% RSLogix 500 project P7_KOBIERSKI_M.RSS, saved by version 8.30.00.16 %
PROJECT "UNTITLED"    % processor: Bul.1763 MicroLogix 1100 Series B %

PROGRAM FILES
  LAD 2 "MAIN"  4 rungs
  LAD 3 "IO"  6 rungs
  LAD 4 "CYCLE"  5 rungs
  LAD 5 "CALIBRATE"  15 rungs
  LAD 6 "SAMPLE"  7 rungs
  LAD 7 "0% SAMPLE"  7 rungs
  LAD 8 "30% SAMPLE"  7 rungs
  LAD 9 "CALIB CALC"  6 rungs

DATA FILES
  O0 OUTPUT  4 elements
  I1 INPUT  6 elements
  S2 STATUS  66 elements
  B3 BINARY  3 elements
  T4 TIMER  5 elements
  C5 COUNTER  1 elements
  R6 CONTROL  1 elements
  N7 INTEGER  9 elements
  F8 FLOAT  3 elements
  F9 O2 SAMPLES  10 elements
  N10 SAMP STTNG  6 elements
  F11 AVGS  9 elements
  F12 0% SAMPLES  5 elements
  F13 30% SAMPLE  5 elements
  F14 CALIB MATH  4 elements

LADDER 2 "MAIN"
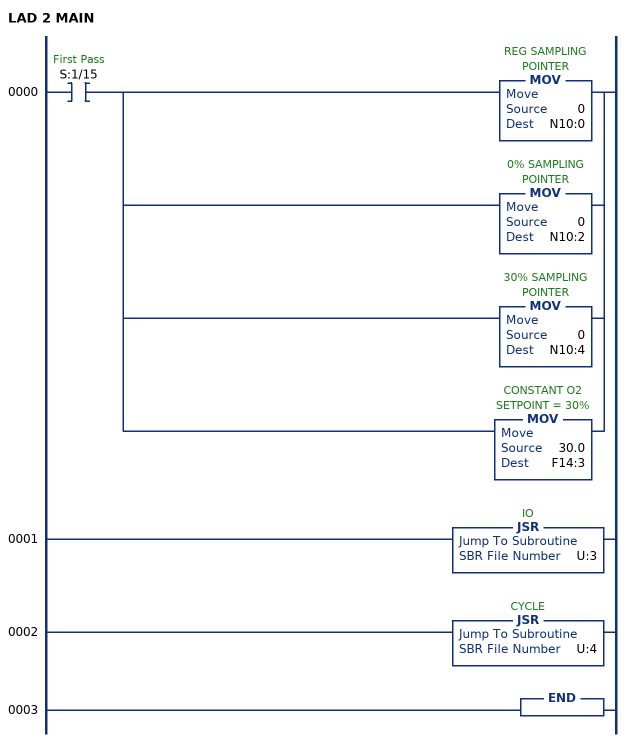
% Rung: 0 %
SOR XIC S:1/15 BST MOV 0 N10:0 NXB MOV 0 N10:2 NXB MOV 0 N10:4 NXB MOV 30.0 F14:3 BND EOR
%   S:1/15  "First Pass" %
%   N10:0  "REG SAMPLING POINTER" %
%   N10:2  "0% SAMPLING POINTER" %
%   N10:4  "30% SAMPLING POINTER" %
%   F14:3  "CONSTANT O2 SETPOINT = 30%" %
% Rung: 1 %
SOR JSR U:3 EOR
%   U:3  "IO" %
% Rung: 2 %
SOR JSR U:4 EOR
%   U:4  "CYCLE" %
% Rung: 3 %
SOR END EOR

LADDER 3 "IO"
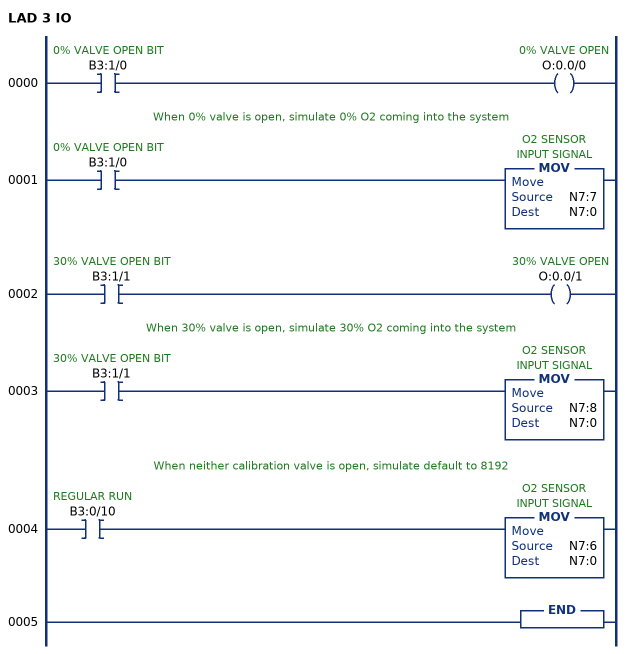
% Rung: 0 %
SOR XIC B3:1/0 OTE O:0.0/0 EOR
%   B3:1/0  "0% VALVE OPEN BIT" %
%   O:0.0/0  "0% VALVE OPEN" %
% Rung: 1 %
% When 0% valve is open, simulate 0% O2 coming into the system %
SOR XIC B3:1/0 MOV N7:7 N7:0 EOR
%   B3:1/0  "0% VALVE OPEN BIT" %
%   N7:7  "SIMULATED 0% SIGNAL" %
%   N7:0  "O2 SENSOR INPUT SIGNAL" %
% Rung: 2 %
SOR XIC B3:1/1 OTE O:0.0/1 EOR
%   B3:1/1  "30% VALVE OPEN BIT" %
%   O:0.0/1  "30% VALVE OPEN" %
% Rung: 3 %
% When 30% valve is open, simulate 30% O2 coming into the system %
SOR XIC B3:1/1 MOV N7:8 N7:0 EOR
%   B3:1/1  "30% VALVE OPEN BIT" %
%   N7:8  "SIMULATED 30% SIGNAL" %
%   N7:0  "O2 SENSOR INPUT SIGNAL" %
% Rung: 4 %
% When neither calibration valve is open, simulate default to 8192 %
SOR XIC B3:0/10 MOV N7:6 N7:0 EOR
%   B3:0/10  "REGULAR RUN" %
%   N7:6  "SIMULATED INPUT SIGNAL" %
%   N7:0  "O2 SENSOR INPUT SIGNAL" %
% Rung: 5 %
SOR END EOR

LADDER 4 "CYCLE"
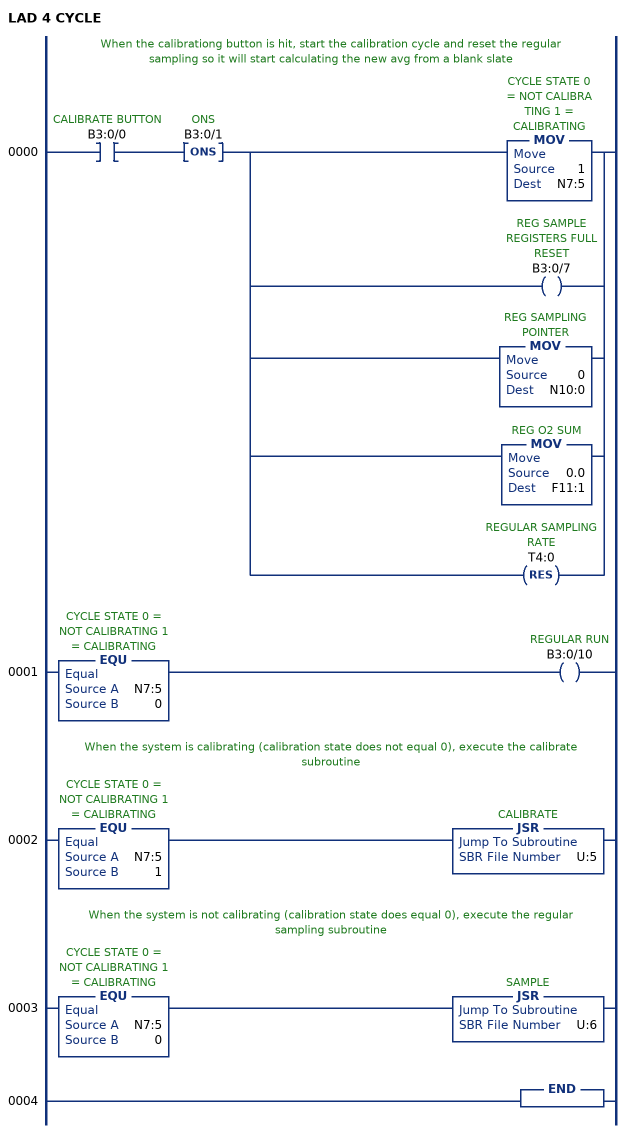
% Rung: 0 %
% When the calibrationg button is hit, start the calibration cycle and reset the regular sampling so it will start calculating the new avg from a blank slate %
SOR XIC B3:0/0 ONS B3:0/1 BST MOV 1 N7:5 NXB OTE B3:0/7 NXB MOV 0 N10:0 NXB MOV 0.0 F11:1 NXB RES T4:0 BND EOR
%   B3:0/0  "CALIBRATE BUTTON" %
%   B3:0/1  "ONS" %
%   N7:5  "CYCLE STATE 0 = NOT CALIBRATING 1 = CALIBRATING" %
%   B3:0/7  "REG SAMPLE REGISTERS FULL RESET" %
%   N10:0  "REG SAMPLING POINTER" %
%   F11:1  "REG O2 SUM" %
%   T4:0  "REGULAR SAMPLING RATE" %
% Rung: 1 %
SOR EQU N7:5 0 OTE B3:0/10 EOR
%   N7:5  "CYCLE STATE 0 = NOT CALIBRATING 1 = CALIBRATING" %
%   B3:0/10  "REGULAR RUN" %
% Rung: 2 %
% When the system is calibrating (calibration state does not equal 0), execute the calibrate subroutine %
SOR EQU N7:5 1 JSR U:5 EOR
%   N7:5  "CYCLE STATE 0 = NOT CALIBRATING 1 = CALIBRATING" %
%   U:5  "CALIBRATE" %
% Rung: 3 %
% When the system is not calibrating (calibration state does equal 0), execute the regular sampling subroutine %
SOR EQU N7:5 0 JSR U:6 EOR
%   N7:5  "CYCLE STATE 0 = NOT CALIBRATING 1 = CALIBRATING" %
%   U:6  "SAMPLE" %
% Rung: 4 %
SOR END EOR

LADDER 5 "CALIBRATE"
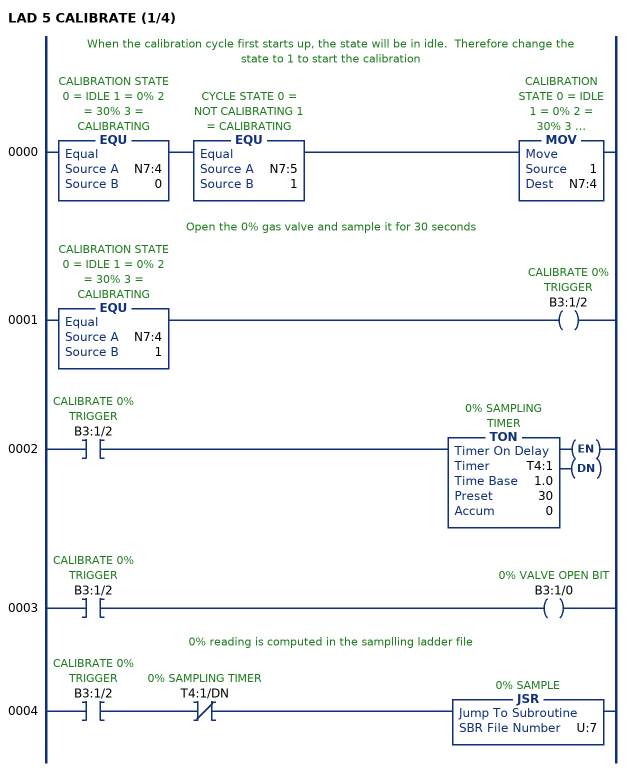
% Rung: 0 %
% When the calibration cycle first starts up, the state will be in idle.  Therefore change the state to 1 to start the calibration %
SOR EQU N7:4 0 EQU N7:5 1 MOV 1 N7:4 EOR
%   N7:4  "CALIBRATION STATE 0 = IDLE 1 = 0% 2 = 30% 3 = CALIBRATING" %
%   N7:5  "CYCLE STATE 0 = NOT CALIBRATING 1 = CALIBRATING" %
% Rung: 1 %
% Open the 0% gas valve and sample it for 30 seconds %
SOR EQU N7:4 1 OTE B3:1/2 EOR
%   N7:4  "CALIBRATION STATE 0 = IDLE 1 = 0% 2 = 30% 3 = CALIBRATING" %
%   B3:1/2  "CALIBRATE 0% TRIGGER" %
% Rung: 2 %
SOR XIC B3:1/2 TON T4:1 1.0 30 0 EOR
%   B3:1/2  "CALIBRATE 0% TRIGGER" %
%   T4:1  "0% SAMPLING TIMER" %
% Rung: 3 %
SOR XIC B3:1/2 OTE B3:1/0 EOR
%   B3:1/2  "CALIBRATE 0% TRIGGER" %
%   B3:1/0  "0% VALVE OPEN BIT" %
% Rung: 4 %
% 0% reading is computed in the samplling ladder file %
SOR XIC B3:1/2 XIO T4:1/DN JSR U:7 EOR
%   B3:1/2  "CALIBRATE 0% TRIGGER" %
%   T4:1  "0% SAMPLING TIMER" %
%   U:7  "0% SAMPLE" %

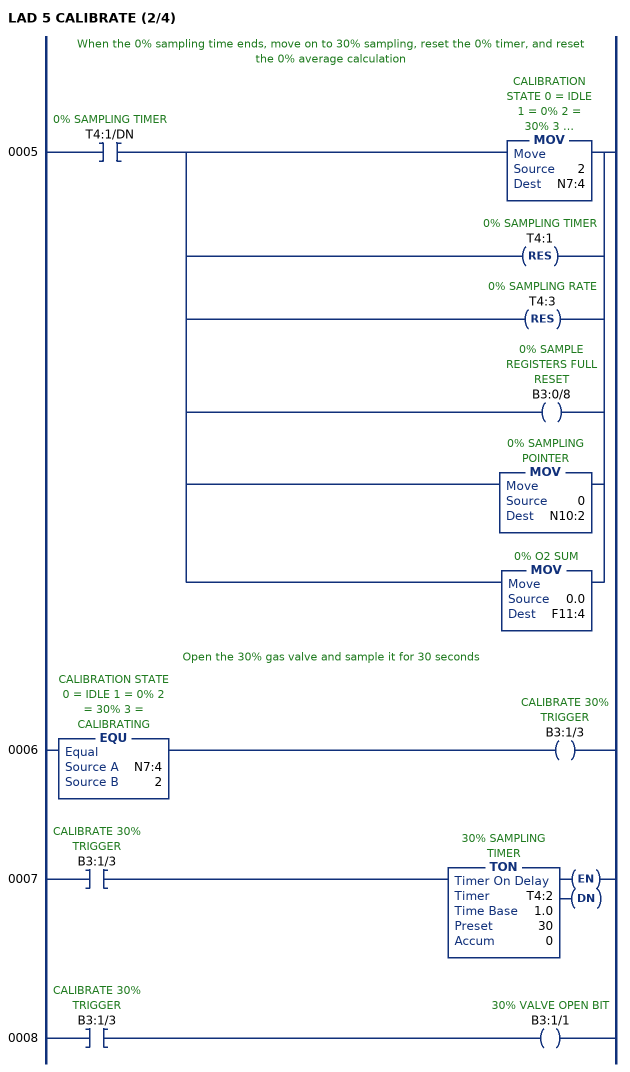
% Rung: 5 %
% When the 0% sampling time ends, move on to 30% sampling, reset the 0% timer, and reset the 0% average calculation %
SOR XIC T4:1/DN BST MOV 2 N7:4 NXB RES T4:1 NXB RES T4:3 NXB OTE B3:0/8 NXB MOV 0 N10:2 NXB MOV 0.0 F11:4 BND EOR
%   T4:1  "0% SAMPLING TIMER" %
%   N7:4  "CALIBRATION STATE 0 = IDLE 1 = 0% 2 = 30% 3 = CALIBRATING" %
%   T4:3  "0% SAMPLING RATE" %
%   B3:0/8  "0% SAMPLE REGISTERS FULL RESET" %
%   N10:2  "0% SAMPLING POINTER" %
%   F11:4  "0% O2 SUM" %
% Rung: 6 %
% Open the 30% gas valve and sample it for 30 seconds %
SOR EQU N7:4 2 OTE B3:1/3 EOR
%   N7:4  "CALIBRATION STATE 0 = IDLE 1 = 0% 2 = 30% 3 = CALIBRATING" %
%   B3:1/3  "CALIBRATE 30% TRIGGER" %
% Rung: 7 %
SOR XIC B3:1/3 TON T4:2 1.0 30 0 EOR
%   B3:1/3  "CALIBRATE 30% TRIGGER" %
%   T4:2  "30% SAMPLING TIMER" %
% Rung: 8 %
SOR XIC B3:1/3 OTE B3:1/1 EOR
%   B3:1/3  "CALIBRATE 30% TRIGGER" %
%   B3:1/1  "30% VALVE OPEN BIT" %

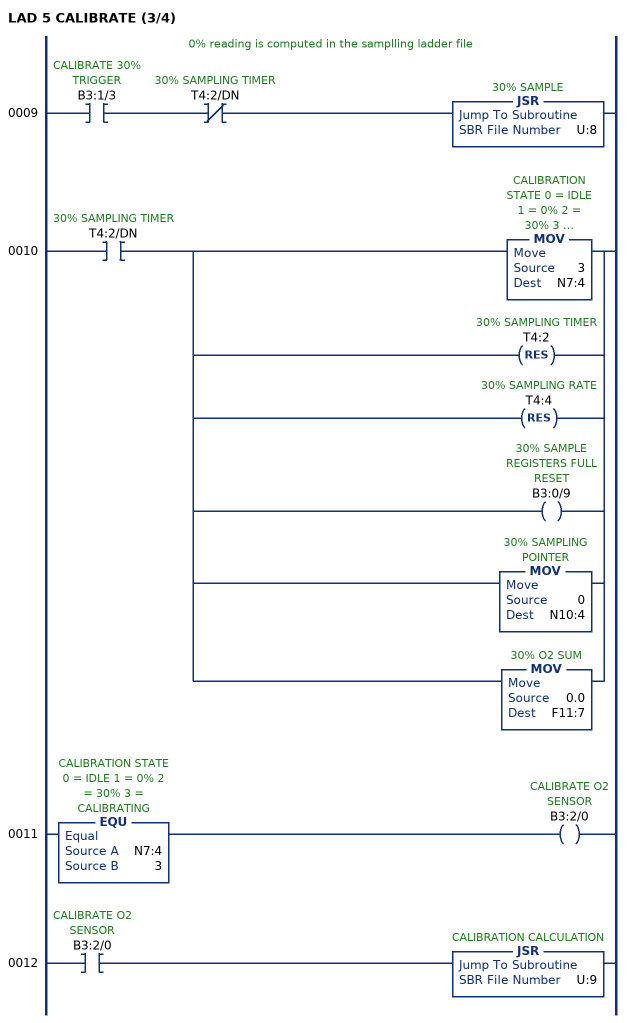
% Rung: 9 %
% 0% reading is computed in the samplling ladder file %
SOR XIC B3:1/3 XIO T4:2/DN JSR U:8 EOR
%   B3:1/3  "CALIBRATE 30% TRIGGER" %
%   T4:2  "30% SAMPLING TIMER" %
%   U:8  "30% SAMPLE" %
% Rung: 10 %
SOR XIC T4:2/DN BST MOV 3 N7:4 NXB RES T4:2 NXB RES T4:4 NXB OTE B3:0/9 NXB MOV 0 N10:4 NXB MOV 0.0 F11:7 BND EOR
%   T4:2  "30% SAMPLING TIMER" %
%   N7:4  "CALIBRATION STATE 0 = IDLE 1 = 0% 2 = 30% 3 = CALIBRATING" %
%   T4:4  "30% SAMPLING RATE" %
%   B3:0/9  "30% SAMPLE REGISTERS FULL RESET" %
%   N10:4  "30% SAMPLING POINTER" %
%   F11:7  "30% O2 SUM" %
% Rung: 11 %
SOR EQU N7:4 3 OTE B3:2/0 EOR
%   N7:4  "CALIBRATION STATE 0 = IDLE 1 = 0% 2 = 30% 3 = CALIBRATING" %
%   B3:2/0  "CALIBRATE O2 SENSOR" %
% Rung: 12 %
SOR XIC B3:2/0 JSR U:9 EOR
%   B3:2/0  "CALIBRATE O2 SENSOR" %
%   U:9  "CALIBRATION CALCULATION" %

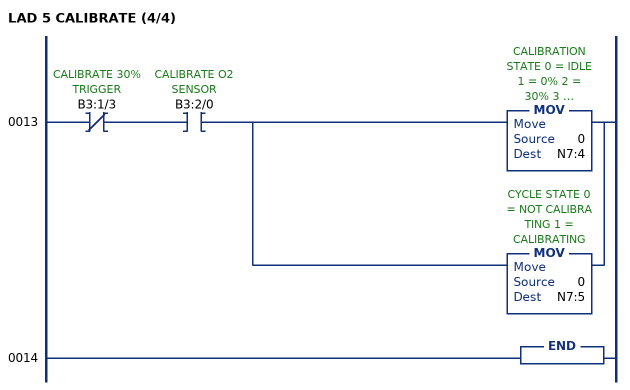
% Rung: 13 %
SOR XIO B3:1/3 XIC B3:2/0 BST MOV 0 N7:4 NXB MOV 0 N7:5 BND EOR
%   B3:1/3  "CALIBRATE 30% TRIGGER" %
%   B3:2/0  "CALIBRATE O2 SENSOR" %
%   N7:4  "CALIBRATION STATE 0 = IDLE 1 = 0% 2 = 30% 3 = CALIBRATING" %
%   N7:5  "CYCLE STATE 0 = NOT CALIBRATING 1 = CALIBRATING" %
% Rung: 14 %
SOR END EOR

LADDER 6 "SAMPLE"
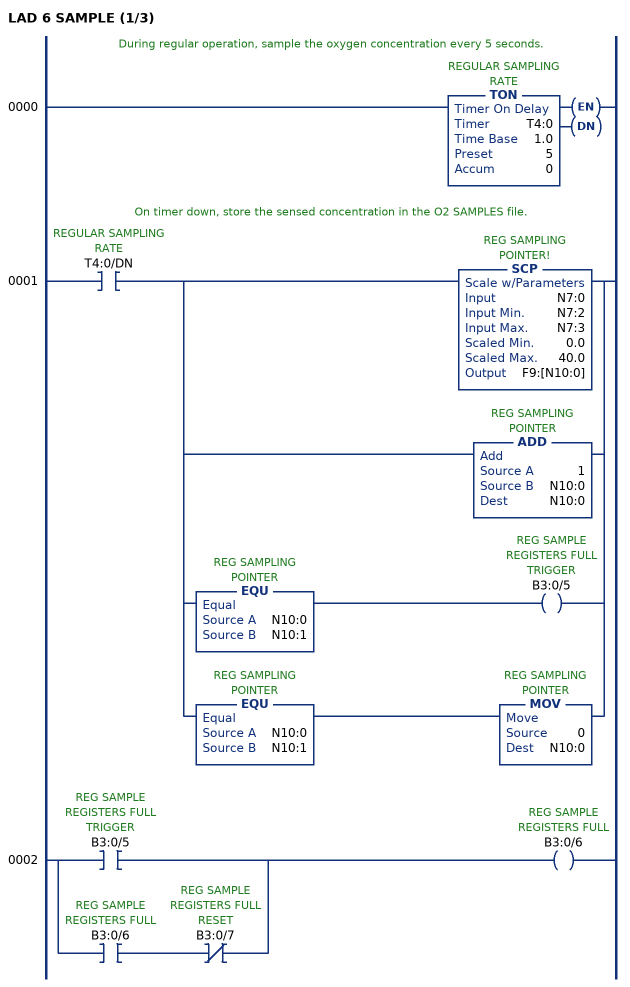
% Rung: 0 %
% During regular operation, sample the oxygen concentration every 5 seconds. %
SOR TON T4:0 1.0 5 0 EOR
%   T4:0  "REGULAR SAMPLING RATE" %
% Rung: 1 %
% On timer down, store the sensed concentration in the O2 SAMPLES file. %
SOR XIC T4:0/DN BST SCP N7:0 N7:2 N7:3 0.0 40.0 F9:[N10:0] NXB ADD 1 N10:0 N10:0 NXB EQU N10:0 N10:1 OTE B3:0/5 NXB EQU N10:0 N10:1 MOV 0 N10:0 BND EOR
%   T4:0  "REGULAR SAMPLING RATE" %
%   N7:0  "O2 SENSOR INPUT SIGNAL" %
%   N7:2  "O2 INPUT MIN" %
%   N7:3  "O2 INPUT MAX" %
%   F9:[N10:0]  "REG SAMPLING POINTER!" %
%   N10:0  "REG SAMPLING POINTER" %
%   N10:1  "REG SAMPLING MAX REGISTERS" %
%   B3:0/5  "REG SAMPLE REGISTERS FULL TRIGGER" %
% Rung: 2 %
SOR BST XIC B3:0/5 NXB XIC B3:0/6 XIO B3:0/7 BND OTE B3:0/6 EOR
%   B3:0/5  "REG SAMPLE REGISTERS FULL TRIGGER" %
%   B3:0/6  "REG SAMPLE REGISTERS FULL" %
%   B3:0/7  "REG SAMPLE REGISTERS FULL RESET" %

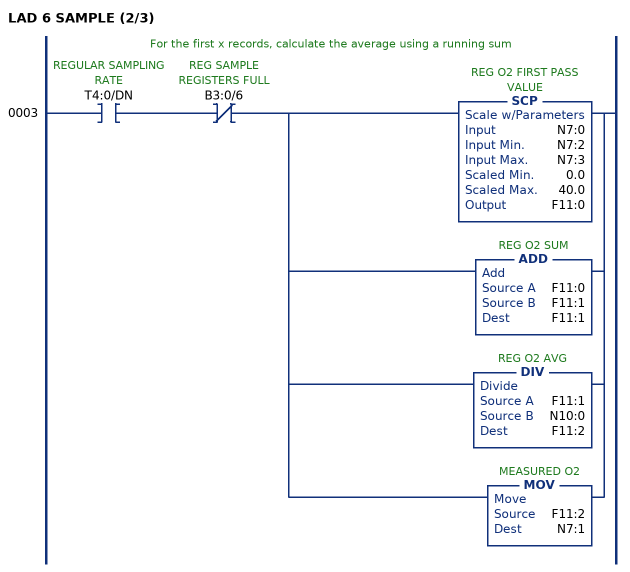
% Rung: 3 %
% For the first x records, calculate the average using a running sum %
SOR XIC T4:0/DN XIO B3:0/6 BST SCP N7:0 N7:2 N7:3 0.0 40.0 F11:0 NXB ADD F11:0 F11:1 F11:1 NXB DIV F11:1 N10:0 F11:2 NXB MOV F11:2 N7:1 BND EOR
%   T4:0  "REGULAR SAMPLING RATE" %
%   B3:0/6  "REG SAMPLE REGISTERS FULL" %
%   N7:0  "O2 SENSOR INPUT SIGNAL" %
%   N7:2  "O2 INPUT MIN" %
%   N7:3  "O2 INPUT MAX" %
%   F11:0  "REG O2 FIRST PASS VALUE" %
%   F11:1  "REG O2 SUM" %
%   N10:0  "REG SAMPLING POINTER" %
%   F11:2  "REG O2 AVG" %
%   N7:1  "MEASURED O2" %

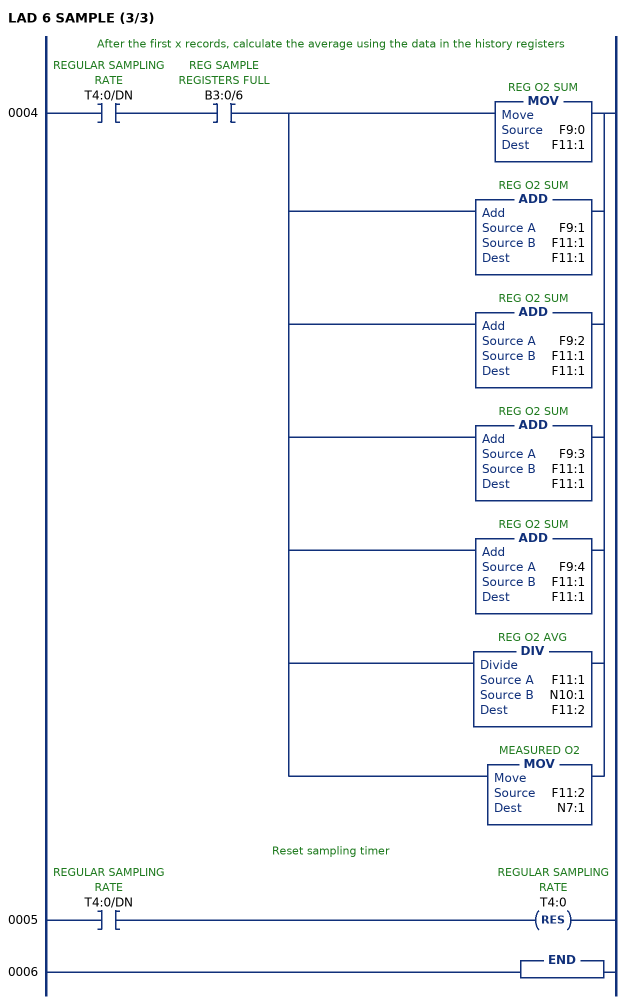
% Rung: 4 %
% After the first x records, calculate the average using the data in the history registers %
SOR XIC T4:0/DN XIC B3:0/6 BST MOV F9:0 F11:1 NXB ADD F9:1 F11:1 F11:1 NXB ADD F9:2 F11:1 F11:1 NXB ADD F9:3 F11:1 F11:1 NXB ADD F9:4 F11:1 F11:1 NXB DIV F11:1 N10:1 F11:2 NXB MOV F11:2 N7:1 BND EOR
%   T4:0  "REGULAR SAMPLING RATE" %
%   B3:0/6  "REG SAMPLE REGISTERS FULL" %
%   F9:0  "O2 SAMPLE AVG" %
%   F11:1  "REG O2 SUM" %
%   F9:1  "O2 SAMPLES" %
%   N10:1  "REG SAMPLING MAX REGISTERS" %
%   F11:2  "REG O2 AVG" %
%   N7:1  "MEASURED O2" %
% Rung: 5 %
% Reset sampling timer %
SOR XIC T4:0/DN RES T4:0 EOR
%   T4:0  "REGULAR SAMPLING RATE" %
% Rung: 6 %
SOR END EOR

LADDER 7 "0% SAMPLE"
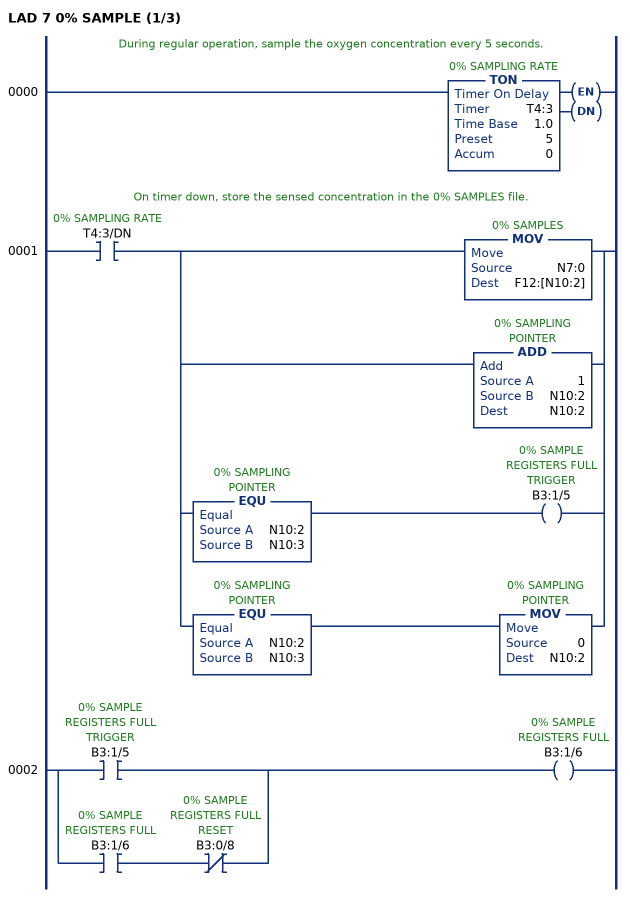
% Rung: 0 %
% During regular operation, sample the oxygen concentration every 5 seconds. %
SOR TON T4:3 1.0 5 0 EOR
%   T4:3  "0% SAMPLING RATE" %
% Rung: 1 %
% On timer down, store the sensed concentration in the 0% SAMPLES file. %
SOR XIC T4:3/DN BST MOV N7:0 F12:[N10:2] NXB ADD 1 N10:2 N10:2 NXB EQU N10:2 N10:3 OTE B3:1/5 NXB EQU N10:2 N10:3 MOV 0 N10:2 BND EOR
%   T4:3  "0% SAMPLING RATE" %
%   N7:0  "O2 SENSOR INPUT SIGNAL" %
%   F12:[N10:2]  "0% SAMPLES" %
%   N10:2  "0% SAMPLING POINTER" %
%   N10:3  "0% SAMPLING MAX REGISTERS" %
%   B3:1/5  "0% SAMPLE REGISTERS FULL TRIGGER" %
% Rung: 2 %
SOR BST XIC B3:1/5 NXB XIC B3:1/6 XIO B3:0/8 BND OTE B3:1/6 EOR
%   B3:1/5  "0% SAMPLE REGISTERS FULL TRIGGER" %
%   B3:1/6  "0% SAMPLE REGISTERS FULL" %
%   B3:0/8  "0% SAMPLE REGISTERS FULL RESET" %

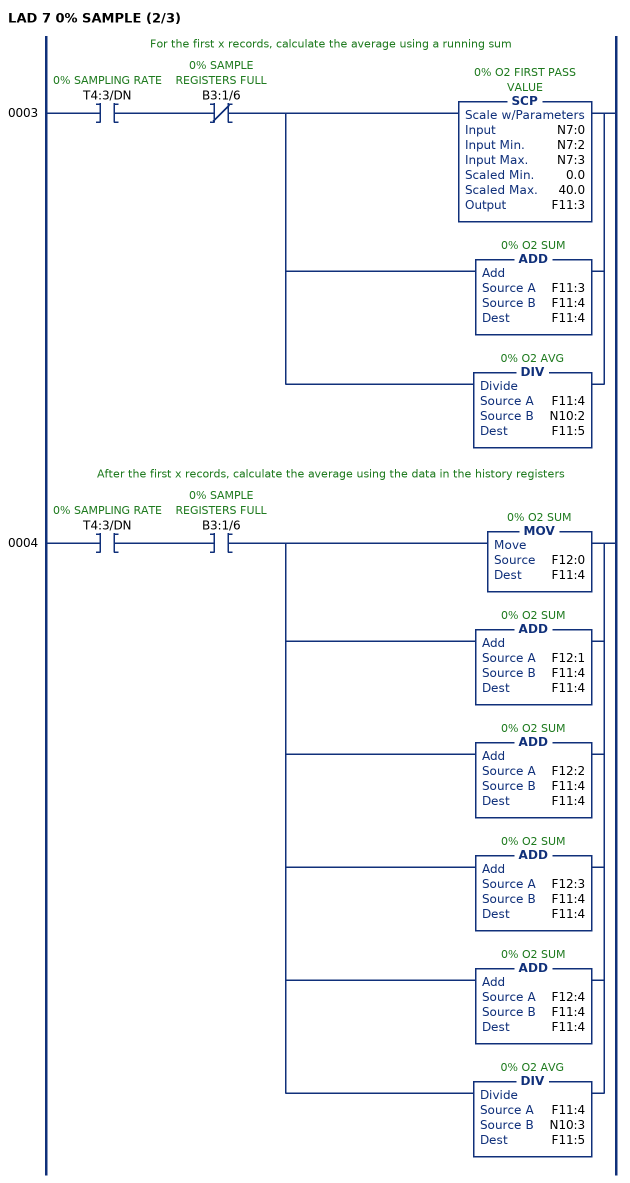
% Rung: 3 %
% For the first x records, calculate the average using a running sum %
SOR XIC T4:3/DN XIO B3:1/6 BST SCP N7:0 N7:2 N7:3 0.0 40.0 F11:3 NXB ADD F11:3 F11:4 F11:4 NXB DIV F11:4 N10:2 F11:5 BND EOR
%   T4:3  "0% SAMPLING RATE" %
%   B3:1/6  "0% SAMPLE REGISTERS FULL" %
%   N7:0  "O2 SENSOR INPUT SIGNAL" %
%   N7:2  "O2 INPUT MIN" %
%   N7:3  "O2 INPUT MAX" %
%   F11:3  "0% O2 FIRST PASS VALUE" %
%   F11:4  "0% O2 SUM" %
%   N10:2  "0% SAMPLING POINTER" %
%   F11:5  "0% O2 AVG" %
% Rung: 4 %
% After the first x records, calculate the average using the data in the history registers %
SOR XIC T4:3/DN XIC B3:1/6 BST MOV F12:0 F11:4 NXB ADD F12:1 F11:4 F11:4 NXB ADD F12:2 F11:4 F11:4 NXB ADD F12:3 F11:4 F11:4 NXB ADD F12:4 F11:4 F11:4 NXB DIV F11:4 N10:3 F11:5 BND EOR
%   T4:3  "0% SAMPLING RATE" %
%   B3:1/6  "0% SAMPLE REGISTERS FULL" %
%   F12:0  "0% SAMPLES" %
%   F11:4  "0% O2 SUM" %
%   N10:3  "0% SAMPLING MAX REGISTERS" %
%   F11:5  "0% O2 AVG" %

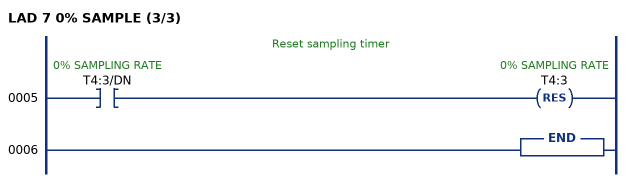
% Rung: 5 %
% Reset sampling timer %
SOR XIC T4:3/DN RES T4:3 EOR
%   T4:3  "0% SAMPLING RATE" %
% Rung: 6 %
SOR END EOR

LADDER 8 "30% SAMPLE"
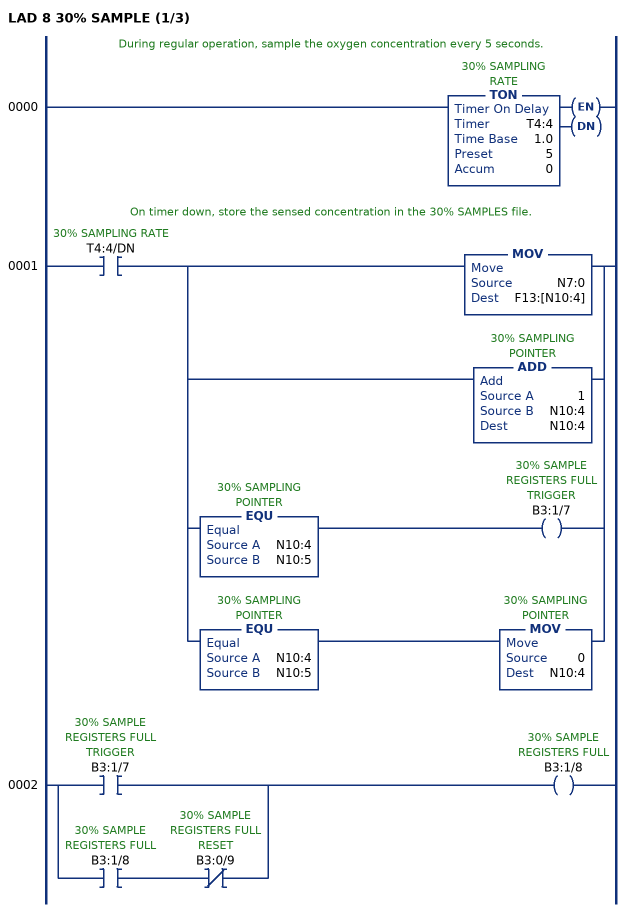
% Rung: 0 %
% During regular operation, sample the oxygen concentration every 5 seconds. %
SOR TON T4:4 1.0 5 0 EOR
%   T4:4  "30% SAMPLING RATE" %
% Rung: 1 %
% On timer down, store the sensed concentration in the 30% SAMPLES file. %
SOR XIC T4:4/DN BST MOV N7:0 F13:[N10:4] NXB ADD 1 N10:4 N10:4 NXB EQU N10:4 N10:5 OTE B3:1/7 NXB EQU N10:4 N10:5 MOV 0 N10:4 BND EOR
%   T4:4  "30% SAMPLING RATE" %
%   N7:0  "O2 SENSOR INPUT SIGNAL" %
%   N10:4  "30% SAMPLING POINTER" %
%   N10:5  "30% SAMPLING MAX REGISTERS" %
%   B3:1/7  "30% SAMPLE REGISTERS FULL TRIGGER" %
% Rung: 2 %
SOR BST XIC B3:1/7 NXB XIC B3:1/8 XIO B3:0/9 BND OTE B3:1/8 EOR
%   B3:1/7  "30% SAMPLE REGISTERS FULL TRIGGER" %
%   B3:1/8  "30% SAMPLE REGISTERS FULL" %
%   B3:0/9  "30% SAMPLE REGISTERS FULL RESET" %

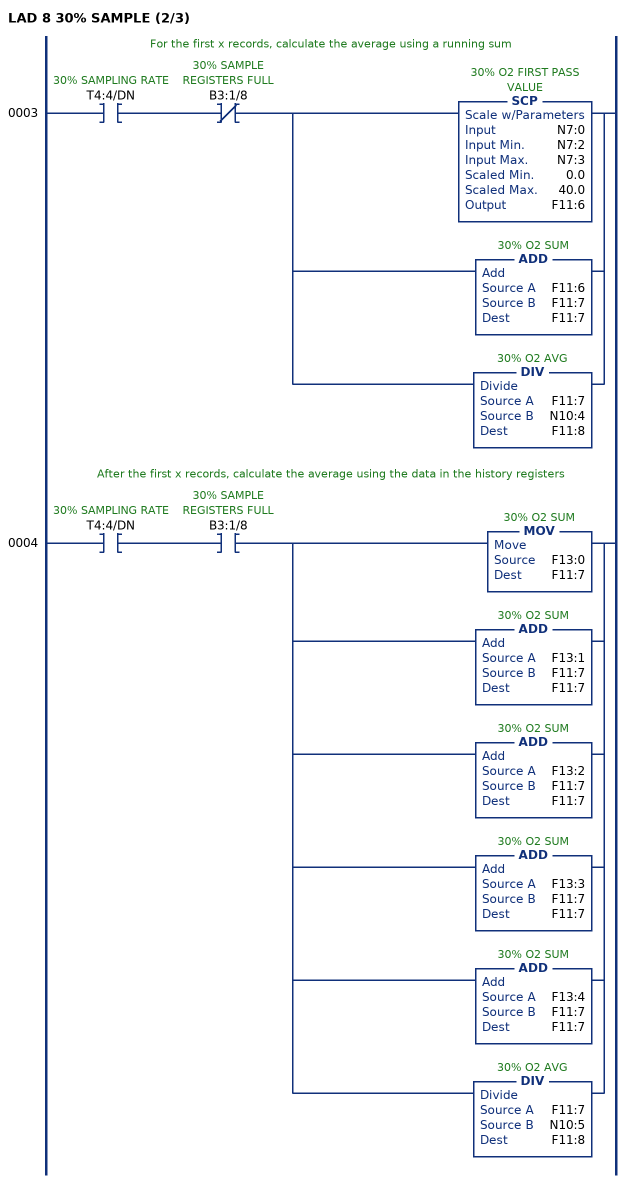
% Rung: 3 %
% For the first x records, calculate the average using a running sum %
SOR XIC T4:4/DN XIO B3:1/8 BST SCP N7:0 N7:2 N7:3 0.0 40.0 F11:6 NXB ADD F11:6 F11:7 F11:7 NXB DIV F11:7 N10:4 F11:8 BND EOR
%   T4:4  "30% SAMPLING RATE" %
%   B3:1/8  "30% SAMPLE REGISTERS FULL" %
%   N7:0  "O2 SENSOR INPUT SIGNAL" %
%   N7:2  "O2 INPUT MIN" %
%   N7:3  "O2 INPUT MAX" %
%   F11:6  "30% O2 FIRST PASS VALUE" %
%   F11:7  "30% O2 SUM" %
%   N10:4  "30% SAMPLING POINTER" %
%   F11:8  "30% O2 AVG" %
% Rung: 4 %
% After the first x records, calculate the average using the data in the history registers %
SOR XIC T4:4/DN XIC B3:1/8 BST MOV F13:0 F11:7 NXB ADD F13:1 F11:7 F11:7 NXB ADD F13:2 F11:7 F11:7 NXB ADD F13:3 F11:7 F11:7 NXB ADD F13:4 F11:7 F11:7 NXB DIV F11:7 N10:5 F11:8 BND EOR
%   T4:4  "30% SAMPLING RATE" %
%   B3:1/8  "30% SAMPLE REGISTERS FULL" %
%   F11:7  "30% O2 SUM" %
%   N10:5  "30% SAMPLING MAX REGISTERS" %
%   F11:8  "30% O2 AVG" %

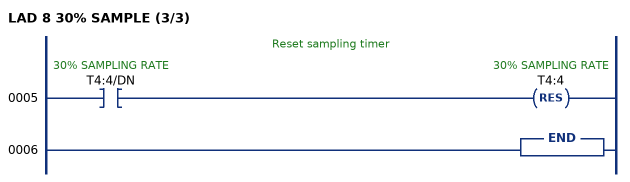
% Rung: 5 %
% Reset sampling timer %
SOR XIC T4:4/DN RES T4:4 EOR
%   T4:4  "30% SAMPLING RATE" %
% Rung: 6 %
SOR END EOR

LADDER 9 "CALIB CALC"
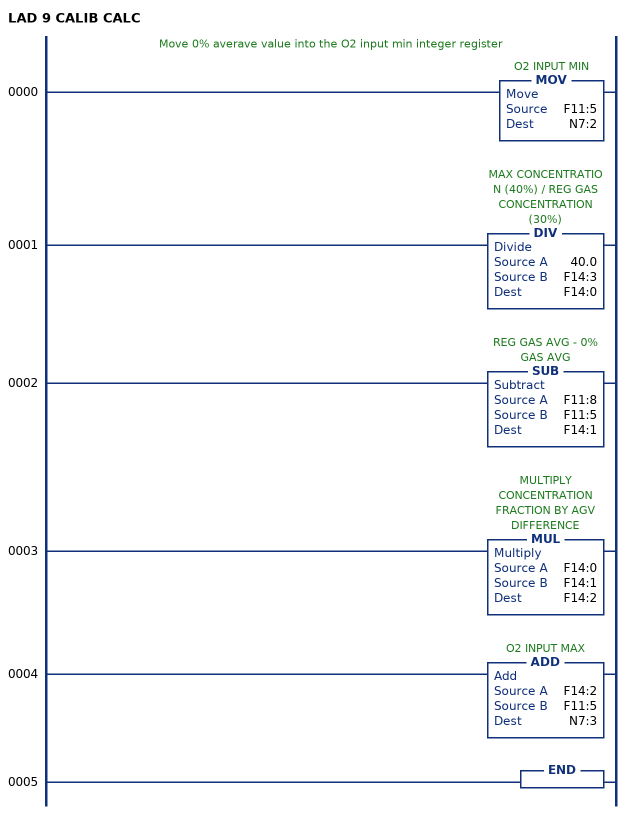
% Rung: 0 %
% Move 0% averave value into the O2 input min integer register %
SOR MOV F11:5 N7:2 EOR
%   F11:5  "0% O2 AVG" %
%   N7:2  "O2 INPUT MIN" %
% Rung: 1 %
SOR DIV 40.0 F14:3 F14:0 EOR
%   F14:3  "CONSTANT O2 SETPOINT = 30%" %
%   F14:0  "MAX CONCENTRATION (40%) / REG GAS CONCENTRATION (30%)" %
% Rung: 2 %
SOR SUB F11:8 F11:5 F14:1 EOR
%   F11:8  "30% O2 AVG" %
%   F11:5  "0% O2 AVG" %
%   F14:1  "REG GAS AVG - 0% GAS AVG" %
% Rung: 3 %
SOR MUL F14:0 F14:1 F14:2 EOR
%   F14:0  "MAX CONCENTRATION (40%) / REG GAS CONCENTRATION (30%)" %
%   F14:1  "REG GAS AVG - 0% GAS AVG" %
%   F14:2  "MULTIPLY CONCENTRATION FRACTION BY AGV DIFFERENCE" %
% Rung: 4 %
SOR ADD F14:2 F11:5 N7:3 EOR
%   F14:2  "MULTIPLY CONCENTRATION FRACTION BY AGV DIFFERENCE" %
%   F11:5  "0% O2 AVG" %
%   N7:3  "O2 INPUT MAX" %
% Rung: 5 %
SOR END EOR

OTHER DOCUMENTED ADDRESSES
  B3:0/2  "CALIBRATE TRIGGER"
  B3:0/3  "CALIBRATE INTERRUPT"
  B3:0/4  "CALIBRATE"
  C5:0  "CALC AVG REG SAMPLE COUNTER"
  F8:0  "REG O2 FIRST PASS DATA"
  F8:1  "REG O2 FIRST PASS RUNNING SUM"
  F8:2  "REG O2 FIRST PASS AVG"
  F9:[F9:0]  "O2 SAMPLE HIST"
  F9:[N7:4]  "REG SAMPLING POINTER"
  N10:0/0  "test"

COMMENTS NOT ATTACHED TO A CURRENT RUNG
  T4:0: During regular operation, sample the oxygen concentration every 5 seconds.
  F11:0: If the registers aren't full, use the counter to sum up all the filled in O2 values
  N7:4: When the calibration cycle first starts up, the state will be in idle.  Therefore change the state to 1 to start the calibration

DATA TABLE (non-zero values as saved)
DATA T4
% .PRE .ACC %
% T4:0 % 5 0
% T4:1 % 30 0
% T4:2 % 30 0
% T4:3 % 5 0
% T4:4 % 5 0
DATA N7
% N7:0 % 8192 0 0 16383 0 0 8192 0 16383
DATA N10
% N10:0 % 0 5 0 5 0 5
